FUNCTION_BLOCK Test_TStreamAdd_Read_BYTE EXTENDS T_UnitTestBase
VAR
    Stream  : T_Stream(StreamLength := 2);
    ArgType : E_ArgTypeId := E_ArgTypeId.Type_BYTE;
END_VAR

{attribute 'analysis' := '-33'} // inhibit unused variable warning
METHOD RunTest
Stream.Init(2);

// add a byte...
Stream.SetNextArgTypeId(ArgType);
Stream.Add_BYTE(123);

Stream.SetReadPosition(0);

// check next arg type is correct...
AssertEquals_INT(Expected     := ArgType,
                           Actual       := Stream.GetNextArgTypeId(),
                           Message := 'Stream.GetNextArgTypeId()');

// check next value...	
AssertEquals_BYTE(Expected     := 123,
                            Actual       := Stream.Read_BYTE(),
                            Message := 'Stream.Read_BYTE()');

// check we are at the end of the stream..							
AssertEquals_UDINT(Expected     := Stream.StreamLength,
                             Actual       := Stream.ReadPosition,
                             Message := 'Stream.ReadPosition');

TestCompleted := TRUE;
END_METHOD

END_FUNCTION_BLOCK

(* stored: Version 1.1.0.1, ProductVersion 3.1.4024.12
   POU Test_TStreamAdd_Read_BYTE: Id {ef58e4d5-752d-42fe-ab45-b9e8aa1637a8}, SpecialFunc None
   Method RunTest: Id {8c4ff1e8-917f-4a6d-bf92-d699f9651967} *)
